// TIA Portal V19 export
TYPE "C301_STU_VEN_TYPIC"
   STRUCT
      CMD { ExternalAccessible := 'False'; ExternalVisible := 'False'; ExternalWritable := 'False'} : USInt;   // Sturing ventilator
      BST { ExternalAccessible := 'False'; ExternalVisible := 'False'; ExternalWritable := 'False'} : USInt;   // Sturing In dienst / Uit dienst
      VGV_BEV { ExternalAccessible := 'False'; ExternalVisible := 'False'; ExternalWritable := 'False'} : USInt;   // Vrijgave ventilator-beveiligingen onbalans en temperatuur
   END_STRUCT;
END_TYPE
